// TIA Portal V17 export
// export: Created 2024-08-09T12:53:16.3414293Z, ExportSetting WithDefaults, DisplayName Totally Integrated Automation Portal, DisplayVersion V17 Update 7, DisplayName TIA Portal Openness, DisplayVersion V17 Update 7, DisplayName TIA Portal Version Control Interface, DisplayVersion V17, DisplayName STEP 7 Professional, DisplayVersion V17 Update 7, DisplayName STEP 7 Safety, DisplayVersion V17 Update 6, DisplayName WinCC Professional, DisplayVersion V17 Update 7
TYPE "S_DECODETRAME"
// stored: IsFailsafeCompliant false
   STRUCT
      KEYWORD : String[20];
      DATA : String;
   END_STRUCT;
END_TYPE
